(* IEC 61131-3 sources: JaccoSigma/tempclass/Class/Carousel, 1 file *)

(* ---- Carousel.st ---- *)
(*!
<Class
	Name               = "Carousel"
	Revision           = "0.0"
	RealtimeTask       = "false"
	CyclicTask         = "false"
	BackgroundTask     = "false"
	Sigmatek           = "false"
	OSInterface        = "false"
	HighPriority       = "false"
	Automatic          = "false"
	UpdateMode         = "Prescan"
	SharedCommandTable = "true"
	Objectsize         = "(300,120)">
	<Channels>
		<Server Name="ClassSvr" Visualized="true" Initialize="false" WriteProtected="false" Retentive="false"/>
	</Channels>
</Class>
*)
Carousel : CLASS
  //Servers:
	ClassSvr 	: SvrChCmd_DINT;
  //Clients:
  //Variables:
  //Functions:
  //Tables:
	FUNCTION @STD
		VAR_OUTPUT
			ret_code	: CONFSTATES;
		END_VAR;
	FUNCTION GLOBAL TAB @CT_;
END_CLASS;
